Yaskawa INFORM job: ARUBA_CYLINDER.JBI

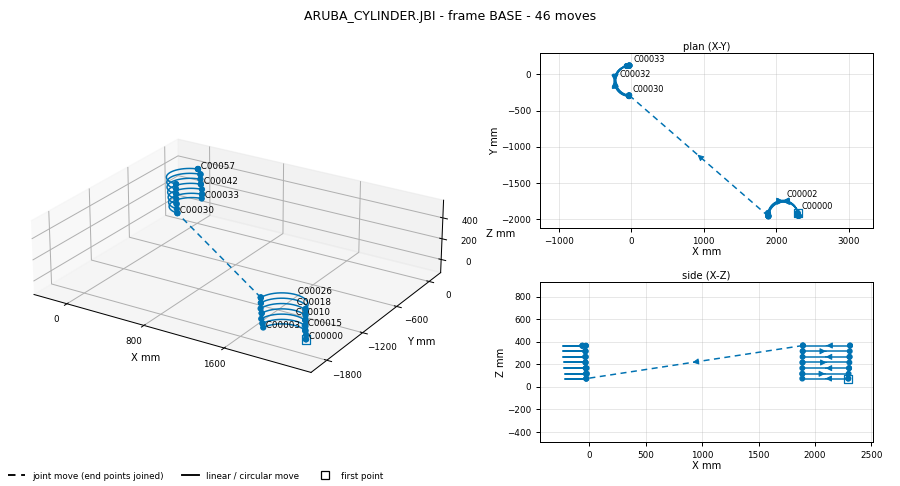
[picture p0: tool path of ARUBA_CYLINDER.JBI in frame BASE, 46 of 66 moves have a stored position in this frame; points joined in program order, loops and branches not executed]
/JOB
//NAME aruba_cylinder_program
//POS
///NPOS 60,0,60,0,0,0
///TOOL 0
///POSTYPE BASE
///RECTAN
///RCONF 0,0,0,0,0,0,0,0,0,0,0,0,0,0,0,0,0,0,0,0,0,0,0,0
C00000=2295.071460,-1910.671304,73.977500,175.000000,-89.999999,5.000000
C00001=2295.071460,-1910.671304,73.977500,175.000000,-89.999999,5.000000
C00002=2094.157113,-1738.356571,73.977500,-90.000000,-90.000000,5.000000
C00003=1887.369145,-1908.592184,73.977500,-0.000000,-89.999999,5.000000
C00004=1887.925283,-1920.965774,116.355000,-0.000000,-89.999999,5.000000
C00005=1887.925283,-1920.965774,116.355000,-0.000000,-89.999999,5.000000
C00006=2073.302923,-1741.536860,116.355000,-90.000000,-90.000000,5.000000
C00007=2297.771372,-1915.110145,116.355000,175.000000,-89.999999,5.000000
C00008=2302.261025,-1938.240952,166.355000,175.000000,-89.999999,5.000000
C00009=2302.261025,-1938.240952,166.355000,175.000000,-89.999999,5.000000
C00010=2074.842048,-1744.807585,166.355000,-90.000000,-90.000000,5.000000
C00011=1887.602772,-1940.475896,166.355000,-0.000000,-89.999999,5.000000
C00012=1889.361535,-1936.929660,216.355000,-0.000000,-89.999999,5.000000
C00013=1889.361535,-1936.929660,216.355000,-0.000000,-89.999999,5.000000
C00014=2083.607565,-1748.964913,216.355000,-90.000000,-90.000000,5.000000
C00015=2304.799047,-1950.615592,216.355000,175.000000,-89.999999,5.000000
C00016=2306.311061,-1947.955535,266.355000,175.000000,-89.999999,5.000000
C00017=2306.311061,-1947.955535,266.355000,175.000000,-89.999999,5.000000
C00018=2086.316552,-1752.373442,266.355000,-90.000000,-90.000000,5.000000
C00019=1889.865912,-1955.282877,266.355000,-0.000000,-89.999999,5.000000
C00020=1891.250862,-1953.235166,316.355000,-0.000000,-89.999999,5.000000
C00021=1891.250862,-1953.235166,316.355000,-0.000000,-89.999999,5.000000
C00022=2083.414835,-1755.770456,316.355000,-90.000000,-90.000000,5.000000
C00023=2308.003776,-1950.138185,316.355000,175.000000,-89.999999,5.000000
C00024=2310.556030,-1953.141011,366.665500,175.000000,-89.999999,5.000000
C00025=2310.556030,-1953.141011,366.665500,175.000000,-89.999999,5.000000
C00026=2101.195846,-1758.877008,366.665500,-90.000000,-90.000000,5.000000
C00027=1892.980848,-1957.672541,366.665500,-0.000000,-89.999999,5.000000
C00028=1892.980848,-1957.672541,366.665500,-0.000000,-89.999999,5.000000
C00029=1892.980848,-1957.672541,366.665500,-0.000000,-89.999999,5.000000
C00030=-27.725453,-288.116460,73.581600,90.000000,-90.000000,5.000000
C00031=-27.725453,-288.116460,73.581600,90.000000,-90.000000,5.000000
C00032=-214.406216,-89.084250,73.581600,5.000000,-89.999999,5.000000
C00033=-27.075286,123.082664,73.581600,-90.000000,-90.000000,5.000000
C00034=-23.426189,123.107631,116.355000,-90.000000,-90.000000,5.000000
C00035=-23.426189,123.107631,116.355000,-90.000000,-90.000000,5.000000
C00036=-218.165683,-70.020956,116.355000,5.000000,-89.999999,5.000000
C00037=-31.534469,-290.372286,116.355000,90.000000,-90.000000,5.000000
C00038=-32.485663,-292.483639,166.355000,90.000000,-90.000000,5.000000
C00039=-32.485663,-292.483639,166.355000,90.000000,-90.000000,5.000000
C00040=-221.735295,-90.451050,166.355000,5.000000,-89.999999,5.000000
C00041=-23.648152,122.179351,166.355000,-90.000000,-90.000000,5.000000
C00042=-33.976186,120.484091,216.355000,-90.000000,-90.000000,5.000000
C00043=-33.976186,120.484091,216.355000,-90.000000,-90.000000,5.000000
C00044=-224.921848,-82.574618,216.355000,5.000000,-89.999999,5.000000
C00045=-33.203318,-294.442376,216.355000,90.000000,-90.000000,5.000000
C00046=-32.549841,-296.547919,266.355000,90.000000,-90.000000,5.000000
C00047=-32.549841,-296.547919,266.355000,90.000000,-90.000000,5.000000
C00048=-230.164118,-96.352434,266.355000,5.000000,-89.999999,5.000000
C00049=-37.748511,119.250390,266.355000,-90.000000,-90.000000,5.000000
C00050=-36.165776,118.346261,316.355000,-90.000000,-90.000000,5.000000
C00051=-36.165776,118.346261,316.355000,-90.000000,-90.000000,5.000000
C00052=-231.046797,-88.838226,316.355000,5.000000,-89.999999,5.000000
C00053=-31.962763,-298.354564,316.355000,90.000000,-90.000000,5.000000
C00054=-30.317620,-299.811099,364.950500,90.000000,-90.000000,5.000000
C00055=-30.317620,-299.811099,364.950500,90.000000,-90.000000,5.000000
C00056=-233.334326,-74.228791,364.950500,5.000000,-89.999999,5.000000
C00057=-61.733838,115.641137,364.950500,-90.000000,-90.000000,5.000000
C00058=-61.733838,115.641137,364.950500,-90.000000,-90.000000,5.000000
C00059=-61.733838,115.641137,364.950500,-90.000000,-90.000000,5.000000
///POSTYPE PULSE
///PULSE
EC00000=0
EC00001=0
EC00002=0
EC00003=0
EC00004=0
EC00005=0
EC00006=0
EC00007=0
EC00008=0
EC00009=0
EC00010=0
EC00011=0
EC00012=0
EC00013=0
EC00014=0
EC00015=0
EC00016=0
EC00017=0
EC00018=0
EC00019=0
EC00020=0
EC00021=0
EC00022=0
EC00023=0
EC00024=0
EC00025=0
EC00026=0
EC00027=0
EC00028=184320
EC00029=368640
EC00030=368640
EC00031=368640
EC00032=368640
EC00033=368640
EC00034=368640
EC00035=368640
EC00036=368640
EC00037=368640
EC00038=368640
EC00039=368640
EC00040=368640
EC00041=368640
EC00042=368640
EC00043=368640
EC00044=368640
EC00045=368640
EC00046=368640
EC00047=368640
EC00048=368640
EC00049=368640
EC00050=368640
EC00051=368640
EC00052=368640
EC00053=368640
EC00054=368640
EC00055=368640
EC00056=368640
EC00057=368640
EC00058=552960
EC00059=737280
//INST
///DATE 2023/05/02 17:32
///ATTR SC,RW,RJ
////FRAME BASE
///GROUP1 RB1,ST1
NOP
MOVJ P009 EX000 VJ=15.00
MOVJ P009 VJ=15.00
MOVJ C00000 EC00000 VJ=15.0
MOVC C00001 EC00001 V=150.0
MOVC C00002 EC00002 V=150.0
MOVC C00003 EC00003 V=150.0
MOVL C00004 EC00004 V=150.0
MOVC C00005 EC00005 V=150.0
MOVC C00006 EC00006 V=150.0
MOVC C00007 EC00007 V=150.0
MOVL C00008 EC00008 V=150.0
MOVC C00009 EC00009 V=150.0
MOVC C00010 EC00010 V=150.0
MOVC C00011 EC00011 V=150.0
MOVL C00012 EC00012 V=150.0
MOVC C00013 EC00013 V=150.0
MOVC C00014 EC00014 V=150.0
MOVC C00015 EC00015 V=150.0
MOVL C00016 EC00016 V=150.0
MOVC C00017 EC00017 V=150.0
MOVC C00018 EC00018 V=150.0
MOVC C00019 EC00019 V=150.0
MOVL C00020 EC00020 V=150.0
MOVC C00021 EC00021 V=150.0
MOVC C00022 EC00022 V=150.0
MOVC C00023 EC00023 V=150.0
MOVL C00024 EC00024 V=150.0
MOVC C00025 EC00025 V=150.0
MOVC C00026 EC00026 V=150.0
MOVC C00027 EC00027 V=150.0
MOVJ P009 VJ=15.00
MOVL C00028 EC00028 V=150.0
MOVJ P009 VJ=15.00
MOVL C00029 EC00029 V=150.0
MOVJ C00030 EC00030 VJ=15.0
MOVC C00031 EC00031 V=150.0
MOVC C00032 EC00032 V=150.0
MOVC C00033 EC00033 V=150.0
MOVL C00034 EC00034 V=150.0
MOVC C00035 EC00035 V=150.0
MOVC C00036 EC00036 V=150.0
MOVC C00037 EC00037 V=150.0
MOVL C00038 EC00038 V=150.0
MOVC C00039 EC00039 V=150.0
MOVC C00040 EC00040 V=150.0
MOVC C00041 EC00041 V=150.0
MOVL C00042 EC00042 V=150.0
MOVC C00043 EC00043 V=150.0
MOVC C00044 EC00044 V=150.0
MOVC C00045 EC00045 V=150.0
MOVL C00046 EC00046 V=150.0
MOVC C00047 EC00047 V=150.0
MOVC C00048 EC00048 V=150.0
MOVC C00049 EC00049 V=150.0
MOVL C00050 EC00050 V=150.0
MOVC C00051 EC00051 V=150.0
MOVC C00052 EC00052 V=150.0
MOVC C00053 EC00053 V=150.0
MOVL C00054 EC00054 V=150.0
MOVC C00055 EC00055 V=150.0
MOVC C00056 EC00056 V=150.0
MOVC C00057 EC00057 V=150.0
MOVJ P009 VJ=15.00
MOVL C00058 EC00058 V=150.0
MOVJ P009 VJ=15.00
MOVL C00059 EC00059 V=150.0
END
